Staubli VAL3: toUppercase.pgx

public program toUppercase(string x_sInput, string& x_sResult)
  local num l_nElement
begin
  x_sResult = ""

  for l_nElement=0 to len(x_sInput)-1
    x_sResult=x_sResult+chr(sel(asc(x_sInput,l_nElement)<97 or asc(x_sInput,l_nElement)>122,asc(x_sInput,l_nElement),asc(x_sInput,l_nElement)-32))
  endFor
end
